FUNCTION_BLOCK FB_SeasonStateMachine EXTENDS FB_StateMachine
VAR
    fbDefaultState:     FB_Default(THIS^, THIS^);
END_VAR

METHOD CurrentSeason : I_SeasonState
VAR_INPUT
END_VAR
__QUERYINTERFACE(THIS^.ipState, CurrentSeason);

IF CurrentSeason = 0 THEN
    CurrentSeason := THIS^.fbDefaultState;
END_IF
END_METHOD

METHOD NextSeason
VAR_INPUT
END_VAR
THIS^.CurrentSeason().NextSeason();
END_METHOD

PROPERTY StateDefault : I_SeasonState
GET
StateDefault := THIS^.fbDefaultState;
END_GET
END_PROPERTY

END_FUNCTION_BLOCK

(* stored: Version 1.1.0.1, ProductVersion 3.1.4024.12
   POU FB_SeasonStateMachine: Id {f7895757-b75c-44d9-8b43-03706a7daad7}, SpecialFunc None
   Method CurrentSeason: Id {108b6707-e2e2-43ee-8eb6-58ef7627d596}
   Method NextSeason: Id {0093a391-4eaa-4329-a094-6217c6317ce6}
   Property StateDefault: Id {3d6eee36-1bc7-4e68-b3af-5da019456c43}
   Get Get: Id {21e03cdb-aa11-43bc-b018-c6698e23bbc2} *)
